KUKA KRL program: palletize.src, palletize.dat

--- palletize.src ---
&ACCESS RVP
&REL 11
&PARAM EDITMASK = *
&PARAM TEMPLATE = C:\KRC\Roboter\Template\vorgabe
&PARAM DISKPATH = KRC:\R1\Program
DEF palletize( )
decl int xx

;Timers
resettimes() ;Accomplishes all three, and stops old advancing timers
;$timer[1]=0 ;palletize
;$timer[2]=0 ;de-palletize
;$timer[3]=0 ;total
;FOLD INI;%{PE}
  ;FOLD BASISTECH INI
    GLOBAL INTERRUPT DECL 3 WHEN $STOPMESS==TRUE DO IR_STOPM ( )
    INTERRUPT ON 3
    BAS (#INITMOV,0 )
  ;ENDFOLD (BASISTECH INI)
;FOLD SPOTTECH INI
USERSPOT(#INIT)
;ENDFOLD (SPOTTECH INI)
;FOLD GRIPPERTECH INI
USER_GRP(0,DUMMY,DUMMY,GDEFAULT)
;ENDFOLD (GRIPPERTECH INI)
  ;FOLD USER INI
    ;Make your modifications here

  ;ENDFOLD (USER INI)
;ENDFOLD (INI)

;FOLD PTP HOME  Vel= 100 % DEFAULT;%{PE}%MKUKATPBASIS,%CMOVE,%VPTP,%P 1:PTP, 2:HOME, 3:, 5:100, 7:DEFAULT
$BWDSTART = FALSE
PDAT_ACT=PDEFAULT
FDAT_ACT=FHOME
BAS (#PTP_PARAMS,100 )
$H_POS=XHOME
PTP  XHOME
;ENDFOLD

;~~~~~~~~~~~~~~~~~~~Calculate Position~~~~~~~~~~~~~~~~~~~~~~

;fold calculate positions

for row = 1 to 4
   for col = 1 to 4
      setdown[row,col] = xstartpos
      setdown[row,col].x = setdown[row,col].x + (row-1)*xoff
      setdown[row,col].y = setdown[row,col].y + (col-1)*yoff
      sstatus[row,col] = setdown[row,col].s
      sturn[row,col] = setdown[row,col].t

      prepos[row,col] = setdown[row,col]
      prepos[row,col].z = prepos[row,col].z + zoff
      pstatus[row,col] = prepos[row,col].s
      pturn[row,col] = prepos[row,col].t
      endfor
   endfor

;manipulate status and turn for specific pre-positions
prepos[3,1].t =27
prepos[4,1].t =27
;endfold

;~~~~~~~~~~~~~~~~~~~Palletize~~~~~~~~~~~~~~~~~~~~~~~~~~~~~~~

;Advance run stop for timer 1
$timer_stop[1] = false
$timer_stop[3] = false

;fold palletize
$out[16] = true
for row = 1 to 4
   for col = 1 to 4
      fetch_block()

      ;set ptp velocity
      for xx = 1 to 6
         $vel_axis[xx] = 75
      endfor

      ;ptp move to prepos
      $tool = tool_data[15]
      $load = load_data[15]
      $base = base_data[1]

      $APO.cdis = 150
      ptp prepos[row,col] c_dis

      ;set the cp velocity 0.3 m/s
      $VEL.cp = 0.3

      lin setdown[row,col]

      opengrip()

      ;set the cp vel 1 m/s
      $VEL.cp = 1

      ;move back to prepos
      lin prepos[row,col] c_dis
      endfor
endfor

wait sec 0
$out[16]=false
$timer_stop[1] = true
$timer[7]=$timer[1]

;endfold


;~~~~~~~~~~~~~~~~~~~De-palletize~~~~~~~~~~~~~~~~~~~~~~~~~~~~

;Advance run stop for timer 1
$timer_stop[2] = false

;fold depalletize

for row = 1 to 4
   for col = 1 to 4

      ;set ptp velocity
      for xx = 1 to 6
         $vel_axis[xx] = 75
      endfor

      ;ptp move to prepos
      $tool = tool_data[15]
      $load = load_data[15]
      $base = base_data[1]

      $APO.cdis = 150
      ptp prepos[row,col] c_dis

      ;set the cp velocity 0.3 m/s
      $VEL.cp = 0.3

      lin setdown[row,col]

      closegrip()

      ;set the cp vel 1 m/s
      $VEL.cp = 1

      ;move back to prepos
      lin prepos[row,col] c_dis

      ;return blocks
      return_block()

      endfor
endfor

;endfold


;FOLD PTP HOME  Vel= 100 % DEFAULT;%{PE}%MKUKATPBASIS,%CMOVE,%VPTP,%P 1:PTP, 2:HOME, 3:, 5:100, 7:DEFAULT
$BWDSTART = FALSE
PDAT_ACT=PDEFAULT
FDAT_ACT=FHOME
BAS (#PTP_PARAMS,100 )
$H_POS=XHOME
PTP  XHOME
;ENDFOLD

wait sec 0
$timer_stop[2] = true
$timer_stop[3] = true
$timer[8]=$timer[2]
$timer[9]=$timer[3]

END

def opengrip()
$out[25] = true
$out[26] = false
$out[14] = true
wait sec 0.25

end

def closegrip()
$out[25] = false
$out[26] = true
$out[14] = false
wait sec 0.25
end

def resettimes()
for ii = 1 to 3
   $timer_stop[ii]=true
   $timer[ii] = 0
endfor
end

--- palletize.dat ---
&ACCESS RVP
&REL 11
&PARAM EDITMASK = *
&PARAM TEMPLATE = C:\KRC\Roboter\Template\vorgabe
&PARAM DISKPATH = KRC:\R1\Program
DEFDAT  palletize
;FOLD EXTERNAL DECLARATIONS;%{PE}%MKUKATPBASIS,%CEXT,%VCOMMON,%P
;FOLD GRIPPERTECH EXT
EXT  H50 (INT  :IN,INT  :IN,INT  :IN,GRP_TYP  :IN )
;ENDFOLD (GRIPPERTECH EXT)
;FOLD SPOTTECH EXT
EXT  USERSPOT (S_COMMAND  :IN,SPOT_TYPE  :IN )
;ENDFOLD (SPOTTECH EXT)
;FOLD BASISTECH EXT;%{PE}%MKUKATPBASIS,%CEXT,%VEXT,%P
EXT  BAS (BAS_COMMAND  :IN,REAL  :IN )
DECL INT SUCCESS
;ENDFOLD (BASISTECH EXT)
;FOLD USER EXT;%{E}%MKUKATPUSER,%CEXT,%VEXT,%P
;Make your modifications here

;ENDFOLD (USER EXT)
;ENDFOLD (EXTERNAL DECLARATIONS)
DECL REAL xoff=80.0000
DECL REAL yoff=80.0000
DECL REAL zoff=100.000

DECL INT row,col,sstatus[4,4],sturn[4,4],pstatus[4,4],pturn[4,4],ii
DECL E6POS prepos[4,4]
prepos[1,1]={X -15.9321737,Y -204.538239,Z 117.342392,A 62.8309174,B 87.5960159,C 62.7038193,S 6,T 58,E1 0.0,E2 0.0,E3 0.0,E4 0.0,E5 0.0,E6 0.0}

DECL E6POS setdown[4,4]
setdown[1,1]={X -15.9321737,Y -204.538239,Z 17.3423920,A 62.8309174,B 87.5960159,C 62.7038193,S 6,T 58,E1 0.0,E2 0.0,E3 0.0,E4 0.0,E5 0.0,E6 0.0}
DECL BASIS_SUGG_T LAST_BASIS={POINT1[] "startpos                ",POINT2[] "startpos                ",CP_PARAMS[] "CPDAT0                  ",PTP_PARAMS[] "PDAT2                   ",CONT[] "                        ",CP_VEL[] "2.0                     ",PTP_VEL[] "100                     ",SYNC_PARAMS[] "SYNCDAT                 ",SPL_NAME[] "S0                      ",A_PARAMS[] "ADAT0                   "}
DECL E6POS XPOUNCE={X 80.9091797,Y -128.856567,Z 172.747818,A 75.6442947,B 86.8682785,C 72.7626724,S 6,T 58,E1 0.0,E2 0.0,E3 0.0,E4 0.0,E5 0.0,E6 0.0}
DECL FDAT Fpounce={TOOL_NO 15,BASE_NO 1,IPO_FRAME #BASE,POINT2[] " ",TQ_STATE FALSE}
DECL PDAT PPDAT1={VEL 100.000,ACC 100.000,APO_DIST 100.000,GEAR_JERK 50.0000,EXAX_IGN 0}
DECL E6POS XSTARTPOS={X -15.9321737,Y -204.538239,Z 17.3423920,A 62.8309174,B 87.5960159,C 62.7038193,S 6,T 58,E1 0.0,E2 0.0,E3 0.0,E4 0.0,E5 0.0,E6 0.0}
DECL FDAT Fstartpos={TOOL_NO 15,BASE_NO 1,IPO_FRAME #BASE,POINT2[] " ",TQ_STATE FALSE}
DECL PDAT PPDAT2={VEL 100.000,ACC 100.000,APO_DIST 100.000,GEAR_JERK 50.0000,EXAX_IGN 0}
ENDDAT
